// TIA Portal V17 export
// export: Created 2022-07-20T06:59:47.3936192Z, ExportSetting WithDefaults, DisplayName Totally Integrated Automation Portal, DisplayVersion V17, DisplayName TIA Portal Openness, DisplayVersion V17, DisplayName TIA Portal Version Control Interface, DisplayVersion V17, DisplayName SINAMICS Startdrive Advanced, DisplayVersion V17, DisplayName SINAMICS Startdrive G130, G150, S120, S150, SINAMICS MV, S210, DisplayVersion V17, DisplayName SINAMICS Startdrive G110M, G120, G120C, G120D, G120P, G115D, DisplayVersion V17, DisplayName STEP 7 Professional, DisplayVersion V17, DisplayName STEP 7 Safety, DisplayVersion V17, DisplayName WinCC Advanced, DisplayVersion V17
FUNCTION_BLOCK "FB10114_OrientalStepperMotorControl"   // FB10114, LAD
TITLE = FB10114_OrientalStepperMotorControl
{ S7_Optimized_Access := 'TRUE' }
AUTHOR : Anirouddh
FAMILY : 1011x_ORIENTAL_MOTOR
VERSION : 1.0
// Release note : 
// 1.0 - Feature developped
// stored: AutoNumber false, IsIECCheckEnabled false, IsRetainMemResEnabled false, MemoryReserve 100, SetENOAutomatically false, UDAEnableTagReadback false
   VAR_INPUT
      HomingSensor : Bool;   // Homing sensor
      OriginPosition : Real;
      WaitingPosition : Real;
      WorkingPosition : Real;
      DegByStep : Real;   // Degree of the motor by step
      ScrewThread : Int;   // Number of mm by turn
      RequestAcknowledge : Bool;
      RequestHoming : Bool;
      RequestGoToOriginPosition : Bool;
      RequestGoToWaitingPosition : Bool;
      RequestGoToWorkingPosition : Bool;
      MotorMoving : Bool;
      PWMCardInError : Bool;
   END_VAR
   VAR_OUTPUT
      PulsesSetPoint : Real;   // Number of pulse for the TM_Pulse function bloc
      MotorDirection : Bool;   // FALSE : Moving towards vertical roller / TRUE : Moving back
      Acknowledge : Bool;
      InitializeMotorCard : Bool;
      DoHoming : Bool;
      GoToOriginPosition : Bool;
      GoToWaitingPosition : Bool;
      GoToWorkingPosition : Bool;
      HomingDone : Bool;   // Homing of the motor is done
      IsInOriginPosition : Bool;
      IsInWaitingPosition : Bool;
      IsInWorkingPosition : Bool;
      MaterialOK : Bool;
   END_VAR
   VAR
      RequestMotorStartUp : Bool;
      MotorStartUpStateDiagram : Int;
      MotorMovementStateDiagram : Int;
      R_TRIG_RequestHoming { S7_SetPoint := 'True'} : R_TRIG;
      R_TRIG_RequestGoToOriginPosition { S7_SetPoint := 'True'} : R_TRIG;
      R_TRIG_RequestGoToWaitingPosition { S7_SetPoint := 'True'} : R_TRIG;
      R_TRIG_RequestGoToWorkingPosition { S7_SetPoint := 'True'} : R_TRIG;
      R_TRIG_HomingSensor { S7_SetPoint := 'True'} : R_TRIG;
      F_TRIG_MotorMoving { S7_SetPoint := 'True'} : F_TRIG;
      TON_GoToOriginPositionSignal { S7_SetPoint := 'True'} : TON_TIME;
      TON_GoToWaitingPositionSignal { S7_SetPoint := 'True'} : TON_TIME;
      TON_GoToWorkingPositionSignal { S7_SetPoint := 'True'} : TON_TIME;
      TON_InitializeMotorCardSignal { S7_SetPoint := 'True'} : TON_TIME;
   END_VAR
   VAR CONSTANT
      WAIT_FOR_MOTOR_START_UP : Int := 0;
      INITIALIZE_POSITION : Int := 10;
      MOTOR_START_UP_DONE : Int := 20;
      "==========" : Bool;
      WAIT_FOR_MOVEMENT_REQUEST : Int := 0;
      HOMING : Int := 10;
      GO_TO_ORIGIN_POSITION : Int := 20;
      GO_TO_WAITING_POSITION : Int := 30;
      GO_TO_WORKING_POSITION : Int := 40;
      INITIALIZE_MOTOR_CARD : Int := 50;
      INITIALIZE_MOTOR_CARD_1 : Int := 60;
      MOVEMENT_DONE : Int := 70;
   END_VAR
BEGIN

REGION Network 1 (SCL): First Scan
   IF "FirstScan" THEN
       #RequestMotorStartUp := TRUE;
       #MaterialOK := FALSE;
       #InitializeMotorCard := FALSE;
       #MotorStartUpStateDiagram := #WAIT_FOR_MOTOR_START_UP;
       #MotorMovementStateDiagram := #WAIT_FOR_MOVEMENT_REQUEST;
   END_IF;
END_REGION

REGION Network 2 (SCL): Edge Signals
   #F_TRIG_MotorMoving(CLK := #MotorMoving);
   #R_TRIG_RequestHoming(CLK := #RequestHoming);
   #R_TRIG_RequestGoToOriginPosition(CLK := #RequestGoToOriginPosition);
   #R_TRIG_RequestGoToWaitingPosition(CLK := #RequestGoToWaitingPosition);
   #R_TRIG_RequestGoToWorkingPosition(CLK := #RequestGoToWorkingPosition);
END_REGION

REGION Network 3 (SCL): Motor Start Up Sequence
   CASE #MotorStartUpStateDiagram OF
       #WAIT_FOR_MOTOR_START_UP:
           IF #RequestMotorStartUp AND #RequestAcknowledge THEN
               #MotorStartUpStateDiagram := #INITIALIZE_POSITION;
           END_IF;
       #INITIALIZE_POSITION:
           #PulsesSetPoint := 5000.0;
           #MotorDirection := FALSE;
           #GoToOriginPosition := TRUE;
           IF #HomingSensor THEN
               //#PulsesSetPoint := 0;
               #GoToOriginPosition := FALSE;
               #Acknowledge := TRUE;
               #IsInOriginPosition := TRUE;
               #IsInWaitingPosition := FALSE;
               #IsInWorkingPosition := FALSE;
               #MotorStartUpStateDiagram := #MOTOR_START_UP_DONE;
           END_IF;
       #MOTOR_START_UP_DONE:
           #MaterialOK := TRUE;
           #RequestMotorStartUp := FALSE;
   END_CASE;
END_REGION

REGION Network 4 (SCL): Motor Movement Management
   CASE #MotorMovementStateDiagram OF
       #WAIT_FOR_MOVEMENT_REQUEST:
           IF #R_TRIG_RequestGoToOriginPosition.Q THEN
               #HomingDone := FALSE;
               #MotorMovementStateDiagram := #GO_TO_ORIGIN_POSITION;
           ELSIF #R_TRIG_RequestGoToWaitingPosition.Q THEN
               #HomingDone := FALSE;
               #MotorMovementStateDiagram := #GO_TO_WAITING_POSITION;
           ELSIF #R_TRIG_RequestGoToWorkingPosition.Q THEN
               #HomingDone := FALSE;
               #MotorMovementStateDiagram := #GO_TO_WORKING_POSITION;
           END_IF;
       #HOMING:
           ;
       #GO_TO_ORIGIN_POSITION:
           IF NOT(#IsInOriginPosition) THEN
               #PulsesSetPoint := 2000.0;
               #MotorDirection := FALSE;
               #GoToOriginPosition := TRUE;
               IF #HomingSensor THEN
                   //#PulsesSetPoint := 0;
                   #GoToOriginPosition := FALSE;
                   #Acknowledge := TRUE;
                   #IsInOriginPosition := TRUE;
                   #IsInWaitingPosition := FALSE;
                   #IsInWorkingPosition := FALSE;
                   IF #TON_GoToOriginPositionSignal.Q THEN
                       #MotorMovementStateDiagram := #MOVEMENT_DONE;
                   END_IF;
               END_IF;
           ELSE
               #IsInOriginPosition := TRUE;
               #IsInWaitingPosition := FALSE;
               #IsInWorkingPosition := FALSE;
               #MotorMovementStateDiagram := #MOVEMENT_DONE;
           END_IF;
       #GO_TO_WAITING_POSITION:
           IF #IsInOriginPosition THEN
               #PulsesSetPoint := #WaitingPosition;
               #MotorDirection := TRUE;
               #GoToWaitingPosition := TRUE;
               IF #F_TRIG_MotorMoving.Q THEN
                   //#PulsesSetPoint := 0;
                   #GoToWaitingPosition := FALSE;
                   #IsInOriginPosition := FALSE;
                   #IsInWaitingPosition := TRUE;
                   #IsInWorkingPosition := FALSE;
                   #MotorMovementStateDiagram := #MOVEMENT_DONE;
               END_IF;
           ELSIF #IsInWorkingPosition THEN
               #PulsesSetPoint := #WorkingPosition - #WaitingPosition;
               #MotorDirection := FALSE;
               #GoToWaitingPosition := TRUE;
               IF #F_TRIG_MotorMoving.Q THEN
                   //#PulsesSetPoint := 0;
                   #GoToWaitingPosition := FALSE;
                   #IsInOriginPosition := FALSE;
                   #IsInWaitingPosition := TRUE;
                   #IsInWorkingPosition := FALSE;
                   #MotorMovementStateDiagram := #MOVEMENT_DONE;
               END_IF;
           ELSE
               #MotorMovementStateDiagram := #MOVEMENT_DONE;
           END_IF;
       #GO_TO_WORKING_POSITION:
           IF #IsInOriginPosition THEN
               #PulsesSetPoint := #WorkingPosition;
               #MotorDirection := TRUE;
               #GoToWorkingPosition := TRUE;
               IF #F_TRIG_MotorMoving.Q THEN
                   //#PulsesSetPoint := 0;
                   #GoToWorkingPosition := FALSE;
                   #IsInOriginPosition := FALSE;
                   #IsInWaitingPosition := FALSE;
                   #IsInWorkingPosition := TRUE;
                   #MotorMovementStateDiagram := #MOVEMENT_DONE;
               END_IF;
           ELSIF #IsInWaitingPosition THEN
               #PulsesSetPoint := #WorkingPosition - #WaitingPosition;
               #MotorDirection := TRUE;
               #GoToWorkingPosition := TRUE;
               IF #F_TRIG_MotorMoving.Q THEN
                   //#PulsesSetPoint := 0;
                   #GoToWorkingPosition := FALSE;
                   #IsInOriginPosition := FALSE;
                   #IsInWaitingPosition := FALSE;
                   #IsInWorkingPosition := TRUE;
                   #MotorMovementStateDiagram := #MOVEMENT_DONE;
               END_IF;
           ELSE
               #MotorMovementStateDiagram := #MOVEMENT_DONE;
           END_IF;
       #INITIALIZE_MOTOR_CARD:
           #PulsesSetPoint := 100;
           #MotorDirection := TRUE;
           #InitializeMotorCard := TRUE;
           IF #F_TRIG_MotorMoving.Q THEN
               #InitializeMotorCard := FALSE;
               #MotorMovementStateDiagram := #INITIALIZE_MOTOR_CARD_1;
           END_IF;
       #INITIALIZE_MOTOR_CARD_1:
           #PulsesSetPoint := 0;
           #MotorDirection := TRUE;
           #InitializeMotorCard := TRUE;
           IF #TON_InitializeMotorCardSignal.Q THEN
               #InitializeMotorCard := FALSE;
               #MotorMovementStateDiagram := #MOVEMENT_DONE;
           END_IF;
       #MOVEMENT_DONE:
           #MotorMovementStateDiagram := #WAIT_FOR_MOVEMENT_REQUEST;
   END_CASE;
END_REGION

REGION Network 5 (SCL): Timer Signals
   //GoToOriginPositionSiganl
   #TON_GoToOriginPositionSignal(IN := #MotorMovementStateDiagram = #GO_TO_ORIGIN_POSITION,
                                 PT := T#2s);

   //GoToWaitingPositionSignal
   #TON_GoToWaitingPositionSignal(IN := #MotorMovementStateDiagram = #GO_TO_WAITING_POSITION,
                                  PT := T#2s);

   //GoToWorkingPositionSignal
   #TON_GoToWorkingPositionSignal(IN := #MotorMovementStateDiagram = #GO_TO_WORKING_POSITION,
                                  PT := T#2s);

   //InitializeMotorCardSignal
   #TON_InitializeMotorCardSignal(IN := (#MotorMovementStateDiagram = #INITIALIZE_MOTOR_CARD) OR (#MotorMovementStateDiagram = #INITIALIZE_MOTOR_CARD_1),
                                  PT := T#200ms);
END_REGION

REGION Network 6 (SCL): Error Managament
   IF #PWMCardInError THEN
       #Acknowledge := TRUE;
   ELSE
       #Acknowledge := FALSE; 
   END_IF;
END_REGION
END_FUNCTION_BLOCK
